// TIA Portal V18 export
DATA_BLOCK "SS1_774A1_16DO_DO_Vars"   // DB11072
{ S7_Optimized_Access := 'FALSE' }
VERSION : 0.1
// stored: AutoNumber false, DBAccessibleFromOPCUA true, IsOnlyStoredInLoadMemory false, IsWriteProtectedInAS false
   VAR
      DO1 { S7_SetPoint := 'True'} : "UDT_DOadv";   // HS Вкл. вн. насос К1 (10.209)
      DO2 { S7_SetPoint := 'True'} : "UDT_DOadv";   // HS Вкл. вн. насос К2 (10.210)
      DO3 { S7_SetPoint := 'True'} : "UDT_DOadv";   // Резерв
      DO4 { S7_SetPoint := 'True'} : "UDT_DOadv";   // HS Дозвіл на роботу котлів
      DO5 { S7_SetPoint := 'True'} : "UDT_DOadv";   // AHU NF Вкл. обігріву пов. засл. (2.202)
      DO6 { S7_SetPoint := 'True'} : "UDT_DOadv";   // Вкл. обігріву дизельпровода (10.211)
      DO7 { S7_SetPoint := 'True'} : "UDT_DOadv";   // Вкл. системи кондиціювання (7.208 + 7.210)
      DO8 { S7_SetPoint := 'True'} : "UDT_DOadv";   // Вкл. тепл. вентилятор (8.215 + 8.216)
      DO9 { S7_SetPoint := 'True'} : "UDT_DOadv";   // Вкл. цирк. насос (8.217)
      DO10 { S7_SetPoint := 'True'} : "UDT_DOadv";   // Резерв
      DO11 { S7_SetPoint := 'True'} : "UDT_DOadv";   // Резерв
      DO12 { S7_SetPoint := 'True'} : "UDT_DOadv";   // Резерв
      DO13 { S7_SetPoint := 'True'} : "UDT_DOadv";   // Резерв
      DO14 { S7_SetPoint := 'True'} : "UDT_DOadv";   // Резерв
      DO15 { S7_SetPoint := 'True'} : "UDT_DOadv";   // Резерв
      DO16 { S7_SetPoint := 'True'} : "UDT_DOadv";   // Резерв
   END_VAR
BEGIN
   DO1.iFuncSystemID := 10;
   DO1.iFuncVar := 10;
   DO2.iFuncSystemID := 10;
   DO2.iFuncVar := 11;
   DO3.iFuncSystemID := 10;
   DO3.iFuncVar := 12;
   DO4.iFuncSystemID := 100;
   DO4.iFuncVar := 1;
   DO5.iFuncSystemID := 100;
   DO5.iFuncVar := 5;
   DO6.iFuncSystemID := 100;
   DO6.iFuncVar := 3;
   DO7.iFuncSystemID := 10;
   DO7.iFuncVar := 5;
   DO8.iFuncSystemID := 10;
   DO8.iFuncVar := 6;
   DO9.iFuncSystemID := 10;
   DO9.iFuncVar := 13;
   DO14.iFuncSystemID := 1;
   DO14.iFuncVar := 1;
   DO14.cMOA := 1;
   DO15.iFuncSystemID := 1;
   DO16.iFuncSystemID := 1;
   DO16.iFuncVar := 3;
END_DATA_BLOCK
